(*
SPDX-FileCopyrightText: © 2026 Oleksandr Tiutyk <trofimich@gmail.com>
SPDX-License-Identifier: MIT
License: https://opensource.org/license/mit
*)

(*!
<summary>Reports a required argument that the caller considers unspecified.</summary>
<description>
The caller detects the invalid argument. Throw records a diagnostic message and source metadata; it does not
inspect the actual argument or decide which types are supported. Dynamic instances belong to the current task
memory manager until cleanup. Dynamic copies are explicitly registered by Clone after construction; plain
__NEW does not transfer ownership to the task manager.
</description>
*)

{attribute 'enable_dynamic_creation'}
{attribute 'no_explicit_call' := 'do not call this function block directly'}
FUNCTION_BLOCK ArgumentNotSpecifiedException EXTENDS GeneralException IMPLEMENTS IArgumentNotSpecifiedException
VAR_STAT
	//! <summary>Class name shared by all instances of this function block.</summary>
	{attribute 'hide'} 
	_ClassName : STRING := __POUNAME();
END_VAR

{attribute 'monitoring' := 'call'}
PROPERTY ClassName : REFERENCE TO STRING
GET
ClassName REF= _ClassName;
END_GET
END_PROPERTY

(*!
<summary>Creates a distinct auto-disposed copy of this concrete exception type.</summary>
<description>
Copies message, code, source and timestamps through CopyGeneralFields; any prepared inner cause remains
borrowed. The current task memory manager owns the clone until cleanup. Allocation failure is terminal.
Descendants with additional payload must override Clone to preserve their type and fields. Registers the newly
constructed instance before copying payload, outside FB_init. Registration failure releases the unregistered
instance and raises a terminal error; copy failure leaves the registered instance owned by the task manager
for cleanup. Custom overrides must follow the same ownership sequence.
</description>
*)
METHOD Clone : IObject
VAR
	exceptionClone : POINTER TO ArgumentNotSpecifiedException;
END_VAR
exceptionClone := __NEW(ArgumentNotSpecifiedException);

IF exceptionClone = 0 THEN
	DynamicMemoryManager.RaiseAllocationFailure();
END_IF

DynamicMemoryManager.RegisterAutoDisposedObject(autoDisposedObject := exceptionClone^);

exceptionClone^.CopyGeneralFields(sourceException := THIS^);

Clone := exceptionClone^;
END_METHOD

(*!
<summary>Provides the library namespace used in diagnostics.</summary>
<description>
Borrowed read-only reference to the compiler-initialized library namespace; no ownership transfer.
</description>
*)
{attribute 'monitoring' := 'call'}
PROPERTY NamespaceName : REFERENCE TO STRING
GET
NamespaceName REF= CurrentNamespace.Name;
END_GET
END_PROPERTY

(*!
<summary>Reports the byte size of this concrete instance.</summary>
<description>
Uses XSIZEOF on the instance. Does not include separately allocated payloads or prove that an arbitrary
address is valid.
</description>
*)
{attribute 'monitoring' := 'call'}
PROPERTY SelfSize : ULINT
GET
SelfSize := XSIZEOF(THIS^);
END_GET
END_PROPERTY

(*!
<summary>Builds the argument diagnostic and propagates this exception.</summary>
<description>
Call in the owning cyclic task, not during FB_init. Captures message, source and timestamps with zero error
code and no inner cause. Supplied names are copied into a local buffer without heap allocation; no caller
storage is retained. Exception clone allocation failure follows the shared terminal memory mechanism.
</description>
<param name="argumentName">Name of the argument rejected by the caller.</param>
*)
METHOD Throw
VAR_INPUT
	sourceNamespaceName : STRING;
	sourceClassName : STRING;
	sourcePOUName : STRING;
	sourcePosition : STRING;
	argumentName : STRING;
END_VAR
VAR
	message : ERROR_MESSAGE;
END_VAR
message := WideStrings.Concat255(
	"Argument '",
	TO_WSTRING(argumentName),
	"' has not specified value in '",
	TO_WSTRING(GetFullPOUName(
		sourceNamespaceName := sourceNamespaceName,
		sourceClassName := sourceClassName,
		sourcePOUName := sourcePOUName
	)),
	"'");

InternalThrow(
	sourceNamespaceName := sourceNamespaceName,
	sourceClassName := sourceClassName,
	sourcePOUName := sourcePOUName,
	sourcePosition := sourcePosition,
	message := message,
	errorCode := 0,
	innerException := 0
);
END_METHOD

END_FUNCTION_BLOCK

(* stored: Version 1.1.0.1
   POU ArgumentNotSpecifiedException: Id {e79a8fac-a833-4981-9da7-5c3a2034721b}, SpecialFunc None
   Property ClassName: Id {79f67f7d-a246-4cbb-8c4a-d748b6b68a8e}
   Get Get: Id {5a21352d-637d-4dfd-893f-a3088862ffcf}
   Method Clone: Id {055e5ef6-23a6-4564-8c4c-f52147ae361d}
   Property NamespaceName: Id {15dbff06-a3f6-450f-be4b-654d0acc8dbd}
   Get Get: Id {51d7c6d3-6aac-4668-a27f-d21be5633f05}
   Property SelfSize: Id {96eb2f70-c595-4960-9edc-a6e217011a12}
   Get Get: Id {35e4e0d4-a3ff-4a73-8a9d-ad87a70ffe89}
   Method Throw: Id {9b786a6c-4933-4e4d-bd9c-5cb0582fdd50} *)
